ABB RobotStudio station: station_layout.rspag

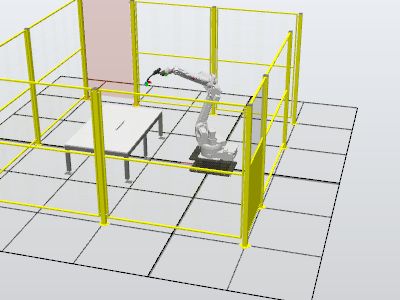
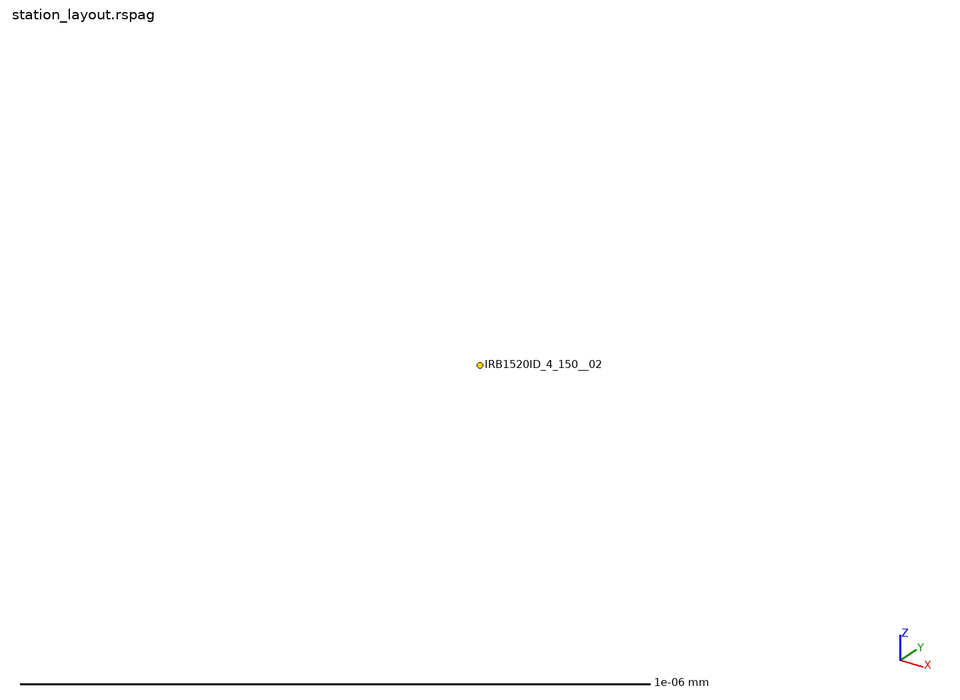
[picture v1: parts stored in the station drawn from their meshes, with robot base, taught points and paths (robot models come from the ABB library and are not in the file)]
--- station ---
Station rdl (saved by RobotStudio 25.5.11605.0)
Controller rdl, task T_ROB1: task frame (RAPID world) sits at (0, 0, 205) mm in the station
Controller rdl
  mechanical unit ROB_1: IRB1520ID_4_150__02, 6 joints, base frame (0, 0, 0) mm
Layout (positions relative to the parent item):
  - RA_MTG4000_22 [mechanism, from %ABB.RobotStudio.Models.ArcWelding%\Fronius_Robacta_MTG4000_22deg.rslib] at (643.33, 235.52, 1605.87) mm, rotated rx -130.29 ry 39.35 rz -118.26 deg
  - IRB1520ID_4_150__02 [mechanism, from %ABB.RobotStudio.Models.IRB1520ID%\IRB1520ID_4_150_G_02.rslib] at (0, 0, 205) mm; joint values [0.4644, -0.3455, -0.1013, -0.4587, 1.0675, -0.27] (rad or m)
  - Robotpedestal1400_H240 [part, from Equipment\Robot Pedestal 1400 H240.rslib] at (-30, 0, 0) mm
  - Fence [graphiccomponentgroup]
    - Segment 1 [part], size 169.7 x 169.7 x 2000 mm
    - Segment 2 [part], size 169.7 x 2056 x 2000 mm
  - Fence_2 [graphiccomponentgroup]
    - Segment 1 [part], size 169.7 x 169.7 x 2000 mm
    - Segment 2 [part], size 1565.8 x 169.7 x 2000 mm
    - Segment 2 [part], size 1565.8 x 169.7 x 2000 mm
  - Fence_3 [graphiccomponentgroup]
    - Segment 1 [part], size 169.7 x 169.7 x 2000 mm
    - Segment 2 [part], size 169.7 x 2076.7 x 2000 mm
    - Segment 2 [part], size 169.7 x 2076.7 x 2000 mm
  - Fence_4 [graphiccomponentgroup]
    - Segment 1 [part], size 169.7 x 169.7 x 2000 mm
    - Segment 2 [part], size 2068.1 x 169.7 x 2000 mm
    - Segment 2 [part], size 2068.1 x 169.7 x 2000 mm
  - Fence_5 [graphiccomponentgroup]
    - Segment 1 [part], size 169.7 x 169.7 x 2000 mm
    - Segment 2 [part], size 169.7 x 1104.5 x 2000 mm
  - Fence_6 [graphiccomponentgroup]
    - Segment 1 [part], size 169.7 x 169.7 x 2000 mm
    - Segment 2 [part], size 169.7 x 1104.5 x 2000 mm
  - Fence_7 [graphiccomponentgroup]
    - Segment 1 [part], size 169.7 x 169.7 x 2000 mm
    - Segment 2 [part], size 169.7 x 1104.5 x 2000 mm
  - Fence_8 [graphiccomponentgroup]
    - Segment 1 [part], size 169.7 x 169.7 x 2000 mm
    - Segment 2 [part], size 1079.7 x 169.7 x 2000 mm
  - Table [part], size 1100 x 1635 x 500 mm
  - A-00677209-00_--E [graphiccomponentgroup] at (1701.18, 200, 677.03) mm, rotated rx 0 ry 0.1 rz 0 deg
    - A-00677226-00.12 [graphiccomponentgroup]
      - P039334634.1 [part], size 32 x 18 x 18 mm
    - A-00677216-00.7 [graphiccomponentgroup]
      - P039334633.2 [part], size 20 x 342 x 30 mm
    - A-00677226-00.11 [graphiccomponentgroup] at (0, 59, 0) mm
      - P039334634.1 [part], size 32 x 18 x 18 mm
Attachment: RA_MTG4000_22 is attached to IRB1520ID_4_150__02 / Link6
Targets, tools, work objects and paths stored in the station and not in the controller backup, written as RAPID:
! task T_ROB1
MODULE CalibData
  PERS tooldata torch:=[TRUE,[[20.31,0,363.689],[0.948464781,0,0.316882565,0]],[1,[0,0,1],[1,0,0,0],0,0,0]];
ENDMODULE


--- Backups/rdl/RAPID/TASK1/PROGMOD/Module1.mod ---
MODULE Module1
    !***********************************************************
    !
    ! Module:  Module1
    !
    ! Description:
    !   <Insert description here>
    !
    ! Author: yassinemac
    !
    ! Version: 1.0
    !
    !***********************************************************


    !***********************************************************
    !
    ! Procedure main
    !
    !   This is the entry point of your program
    !
    !***********************************************************
    PROC main()
        !Add your code here
    ENDPROC
ENDMODULE

--- Backups/rdl/SYSPAR/EIO.cfg ---
EIO:CFG_1.0:6:1::
#
INDUSTRIAL_NETWORK:

      -Name "PROFIBUS" -Label "PROFIBUS Controller Network"\
      -CfgPath "HOME/pbus_cfg.bin"

      -Name "PROFINET" -Connection "PROFINET Network"\
      -Label "PROFINET Controller/Device Network" -StationName ""
#
EIO_CROSS:

      -Name "Arc_1_R1_siR1StopProc" -Res "siR1StopProc" -Act1 "soR1StopProc"

      -Name "Arc_1_R1_siR1ArcEst" -Res "siR1ArcEst" -Act1 "soR1WeldOn"\
      -Oper1 "AND" -Act2 "soR1WeldError" -Act2_invert

      -Name "Arc_1_R1_siR1WaterOk" -Res "siR1WaterOk" -Act1 "soR1WaterError"\
      -Act1_invert

      -Name "Arc_1_R1_siR1GasOk" -Res "siR1GasOk" -Act1 "soR1GasError"\
      -Act1_invert
#
PROFINET_DRIVER:

      -Name "PROFINET_COMMON_DATA"
#
PROFINET_INTERNAL_DEVICE:

      -Name "PN_Internal_Device" -VendorName "ABB Robotics"\
      -ProductName "PROFINET Internal Device"
#
EIO_SIGNAL:

      -Name "siR1StopProc" -SignalType "DI" -Label "Simulated Welder R1"\
      -DeviceMap "0" -Category "Arc_1_R1"

      -Name "siR1ArcEst" -SignalType "DI" -Label "Simulated Welder R1"\
      -DeviceMap "1" -Category "Arc_1_R1"

      -Name "siR1WaterOk" -SignalType "DI" -Label "Simulated Welder R1"\
      -DeviceMap "2" -Category "Arc_1_R1"

      -Name "siR1GasOk" -SignalType "DI" -Label "Simulated Welder R1"\
      -DeviceMap "3" -Category "Arc_1_R1"

      -Name "soR1GasOn" -SignalType "DO" -Label "Simulated Welder R1"\
      -DeviceMap "0" -Category "Arc_1_R1"

      -Name "soR1WeldOn" -SignalType "DO" -Label "Simulated Welder R1"\
      -DeviceMap "1" -Category "Arc_1_R1"

      -Name "soR1FeedOn" -SignalType "DO" -Label "Simulated Welder R1"\
      -DeviceMap "2" -Category "Arc_1_R1"

      -Name "soR1StopProc" -SignalType "DO" -Label "Simulated Welder R1"\
      -DeviceMap "3" -Category "Arc_1_R1" -Access "ALL"

      -Name "soR1WeldError" -SignalType "DO" -Label "Simulated Welder R1"\
      -DeviceMap "4" -Category "Arc_1_R1" -Access "ALL"

      -Name "soR1WaterError" -SignalType "DO" -Label "Simulated Welder R1"\
      -DeviceMap "5" -Category "Arc_1_R1" -Access "ALL"

      -Name "soR1GasError" -SignalType "DO" -Label "Simulated Welder R1"\
      -DeviceMap "6" -Category "Arc_1_R1" -Access "ALL"

      -Name "saoR1Voltage" -SignalType "AO" -Label "Simulated Welder R1"\
      -DeviceMap "17-28" -Category "Arc_1_R1" -EncType "UNSIGNED" -MaxLog 100\
      -MaxPhys 10 -MaxPhysLimit 10 -MaxBitVal 4095

      -Name "saoR1Wirefeed" -SignalType "AO" -Label "Simulated Welder R1"\
      -DeviceMap "17-28" -Category "Arc_1_R1" -EncType "UNSIGNED" -MaxLog 0.5\
      -MaxPhys 10 -MaxPhysLimit 10 -MaxBitVal 4095

--- Backups/rdl/SYSPAR/PROC.cfg ---
PROC:CFG_1.0:6:0::
#
ARC_SYSTEM:

      -name "ARC1" -use_arc_sys_prop "ARC1" -use_arc_err_hndl "default"
#
ARC_SYSTEM_PROP:

      -name "ARC1" -units "SI_UNITS" -use_arc_ui_masking "default"
#
ARC_ROB_PROP:

      -name "ARC1_T_ROB1" -units "SI_UNITS" -scrape_opt_on
#
ARC_ERR_HNDL:

      -name "default" -use_arc_recovery_menu "default"\
      -use_arc_repair_prop "default" -Enabled
#
ARC_RECOVERY_MENU:

      -name "default" -HideAbort
#
ARC_REPAIR_PROP:

      -name "default" -NoRetries 1
#
ARC_UI_MASKING:

      -name "default" -uses_voltage  -uses_wirefeed
#
ARC_EQUIP_CLASS:

      -name "ARC1_EQUIP_T_ROB1" -welder_type "Simulated Welder"\
      -loaded_in_robot "T_ROB1" -use_arc_equip_int "SimWeld_T_ROB1"\
      -use_arc_equip_prop "SimWeld_T_ROB1"
#
ARC_EQUIP_INT:

      -name "SimWeld_T_ROB1" -arc_eq_class "awEquipSTD"\
      -path "RELEASE:/options/arc/WeldEquip/Code/"
#
ARC_EQUIP_PROP:

      -name "SimWeld_T_ROB1" -use_arc_equip_io_di "SimWeld_T_ROB1"\
      -use_arc_equip_io_do "SimWeld_T_ROB1"\
      -use_arc_equip_io_ao "SimWeld_T_ROB1"\
      -use_arc_equip_io_ai "SimWeld_T_ROB1"\
      -use_arc_equip_io_go "SimWeld_T_ROB1"
#
ARC_EQUIP_IO_DI:

      -name "SimWeld_T_ROB1" -StopProc "siR1StopProc" -ArcEst "siR1ArcEst"\
      -ArcEstLabel "MAJOR" -WaterOk "siR1WaterOk" -WaterOkLabel "MAJOR"\
      -GasOk "siR1GasOk" -GasOkLabel "MAJOR"
#
ARC_EQUIP_IO_DO:

      -name "SimWeld_T_ROB1" -GasOn "soR1GasOn" -WeldOn "soR1WeldOn"\
      -FeedOn "soR1FeedOn"
#
ARC_EQUIP_IO_AO:

      -name "SimWeld_T_ROB1" -VoltReference "saoR1Voltage"\
      -FeedReference "saoR1Wirefeed"
#
ARC_EQUIP_IO_AI:

      -name "SimWeld_T_ROB1"
#
ARC_EQUIP_IO_GO:

      -name "SimWeld_T_ROB1"
